TYPE StepperPOSControl :
STRUCT
	Execute : BOOL;
	EmergencyStop : BOOL;
	TargetPosition : UDINT;
	Velocity : INT;
	StartType : UINT;
	Acceleration : UINT;
	Deceleration : UINT;
END_STRUCT
END_TYPE

(* stored: Version 1.1.0.1, ProductVersion 3.1.4024.9
   DUT StepperPOSControl: Id {6e209e3a-24dc-4554-802d-cf4a97ced5aa} *)
